// TIA Portal V19 export
FUNCTION_BLOCK "LAxisCtrlApcFr_UnpubGetCamStatusWord"   // FB19516, LAD
{ S7_Optimized_Access := 'TRUE' }
// stored: IsIECCheckEnabled true, MemoryReserve 100, SetENOAutomatically true
   VAR_INPUT
      Cam { ExternalAccessible := 'False'; ExternalVisible := 'False'; ExternalWritable := 'False'} : DB_ANY;
   END_VAR
   VAR_OUTPUT
      camUsed { ExternalAccessible := 'False'; ExternalVisible := 'False'; ExternalWritable := 'False'} : Bool;
      error { ExternalAccessible := 'False'; ExternalVisible := 'False'; ExternalWritable := 'False'} : Bool;
      restartActive { ExternalAccessible := 'False'; ExternalVisible := 'False'; ExternalWritable := 'False'} : Bool;
      onlineStartValuesChanged { ExternalAccessible := 'False'; ExternalVisible := 'False'; ExternalWritable := 'False'} : Bool;
      camDataChange { ExternalAccessible := 'False'; ExternalVisible := 'False'; ExternalWritable := 'False'} : Bool;
      interpolated { ExternalAccessible := 'False'; ExternalVisible := 'False'; ExternalWritable := 'False'} : Bool;
      interpolation { ExternalAccessible := 'False'; ExternalVisible := 'False'; ExternalWritable := 'False'} : Bool;
   END_VAR
   VAR
      statCam { ExternalAccessible := 'False'; ExternalVisible := 'False'; ExternalWritable := 'False'} : DB_ANY;
      statCamType { ExternalAccessible := 'False'; ExternalVisible := 'False'; ExternalWritable := 'False'} : Int;   // Type of cam
   END_VAR
   VAR CONSTANT
      INVALID_CAM : Int := -3;   // Invalid cam
      CAM_1K : Int := 1;   // Cam type: Cam
      CAM_10K : Int := 2;   // Cam type: Cam_10k
      ERROR_INVALID_TECHNOLOGY_OBJECT : Word := 16#8002;   // See corresponding parameter of MC_ instruction in TIA Portal help (information system)
   END_VAR
BEGIN

REGION Network 1 (SCL)
   //==========================================================================================
   // SIEMENS AG
   // (c)Copyright 2017 All Rights Reserved
   //------------------------------------------------------------------------------------------
   // Library: LAxisCtrl
   // Tested with: S7-1515T-2 PN
   // Engineering: TIA Portal V16
   // Restrictions: ---
   // Requirements: S7-1500/S7-1500T FW 2.5
   // Functionality: Get information from status word
   //------------------------------------------------------------------------------------------
   // Change log table:
   // Version    Date          Expert in charge    Changes applied
   // 01.00.01   23.06.2020    APC                 First released version
   //===========================================================================================

   CASE TypeOfDB(#Cam) OF
       TO_Cam:
           #statCam := #Cam;
           #statCamType := #CAM_1K;

       TO_Cam_10k:
           #statCam := #Cam;
           #statCamType := #CAM_10K;

       ELSE
           #statCam := 0;
           #statCamType := #INVALID_CAM;
   END_CASE;


   CASE #statCamType OF
       #CAM_1K:
           "LAxisCtrlApcFr_UnpubMC_GetCamStatusWord1k"(cam:=#statCam,
                                                       camUsed=>#camUsed,
                                                       error=>#error,
                                                       restartActive=>#restartActive,
                                                       onlineStartValuesChanged=>#onlineStartValuesChanged,
                                                       camDataChange=>#camDataChange,
                                                       interpolated=>#interpolated,
                                                       interpolation=>#interpolation);

       #CAM_10K:
           "LAxisCtrlApcFr_UnpubMC_GetCamStatusWord10k"(cam := #statCam,
                                                       camUsed => #camUsed,
                                                       error => #error,
                                                       restartActive => #restartActive,
                                                       onlineStartValuesChanged => #onlineStartValuesChanged,
                                                       camDataChange => #camDataChange,
                                                       interpolated => #interpolated,
                                                       interpolation => #interpolation);
      #INVALID_CAM:
          #camUsed := FALSE;
          #error := FALSE;
          #restartActive := FALSE;
          #onlineStartValuesChanged := FALSE;
          #camDataChange := FALSE;
          #interpolated := FALSE;
          #interpolation := FALSE;
   END_CASE;
END_REGION
END_FUNCTION_BLOCK
